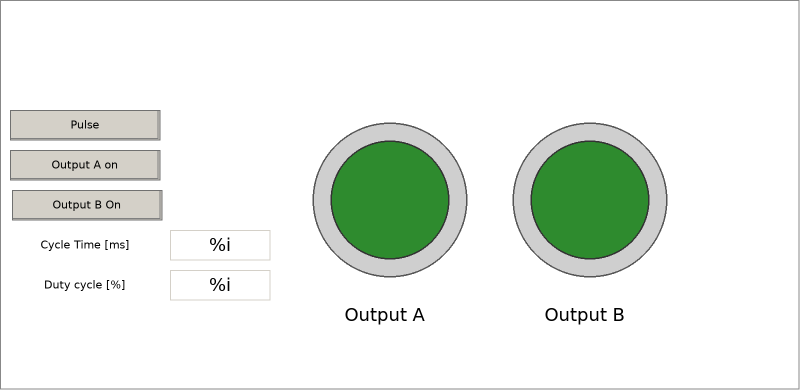
VISUALIZATION VisuDoublePWMControl  // 800x390
    Lamp1 (300,110 180x180), variable: GVL_DevManual.fbManualControler.pDevDoublePWM^.qbOutputA, style: Lamp-Lamp1-Green
    Button (10,110 150x30), "Pulse"
        toggle GVL_DevManual.fbManualControler.pDevDoublePWM^.bCmdPWMOn
    Button (10,150 150x30), "Output A on"
        toggle GVL_DevManual.fbManualControler.pDevDoublePWM^.bCmdChanelAOn
    Textfield (170,230 100x30), "%i", text variable: GVL_DevManual.fbManualControler.pDevDoublePWM^.stParPeriodLength.fValue
        OnMouseUp: write the text variable via VisuDialogs.Numpad
    Label (10,230 150x30), "Cycle Time [ms]"
    Label (10,270 150x30), "Duty cycle [%]"
    Textfield (170,270 100x30), "%i", text variable: GVL_DevManual.fbManualControler.pDevDoublePWM^.stParDutyCycle.fValue
        OnMouseClick: write the text variable via VisuDialogs.Numpad, min 0, max 100
    Lamp1 (500,110 180x180), variable: GVL_DevManual.fbManualControler.pDevPWMController^.qbOutput, style: Lamp-Lamp1-Green
    Button (12,190 150x30), "Output B On"
        tap GVL_DevManual.fbManualControler.pDevDoublePWM^.bCmdChanelBOn
    Label (310,300 150x30), "Output A"
    Label (510,300 150x30), "Output B"
END_VISUALIZATION

(* stored: Version 1.1.0.1, ProductVersion 3.1.4024.5
   Visu VisuDoublePWMControl: Id {df21c097-7ac8-46ed-8ae7-80a53f53d8c0} *)
